KUKA KRL program: centerline_weld.src

&ACCESS RVO1
&REL 38
&COMMENT 03-10-R1 PNW1 NUT WELD
&PARAM TEMPLATE = C:\KRC\Roboter\Template\vorgabe
DEF CENTERLINE_WELD()
;********************************
; Gestamp Standards
; Line - BMW G65 (cell 03)
; Robot 03-10-R1 (BMW-03-10-R1-PNW1)
; Application - NUT WELD AT CENTERLINE PEDESTAL (ALL 3 NUTS)
;********************************
; PRODUCTION NUT WELD, CALLED BY style1app1opt1A..3B OUTSIDE DRY CYCLE WITH THE PART ALREADY
; AT THE WELD POSITION (NO ROBOT MOTION HERE): PEDESTAL START POSITION, UPPER PIN EXTEND,
; PART CLAMP CLOSE, GUN CLOSE, GUN STROKE CHECK (LPT), INTENSIFY, BOSCH WELD; THEN GUN
; OPEN, UPPER PIN RETRACT, PART CLAMP OPEN, LOWER PIN ADVANCE, QFP RETURN.
;WARNING: PEDESTAL ENTRY IS ONLY PARTLY CONFIRMED. THE CALLER CHECKS GUN OPEN (GUN_OPEN_CHECK) AND
;  MONITORS IT WITH INTERRUPTS 20-22; CLAMP OPEN AND QFP RETURNED ARE CHECKED BELOW ONLY AFTER THE
;  ROBOT IS ALREADY AT THE WELD POSITION (F01)
;NOTE: THE NUT IS NORMALLY PRELOADED BY PRELOAD() IN THE SUBMIT INTERPRETER (NUT_READY TRUE);
;  PRELOAD DRIVES THE SAME PEDESTAL VALVES, WITH NO OWNERSHIP BETWEEN THE TWO (F11)
;NOTE: DURING THIS WELD A FEED-ONLY PRELOAD STARTED BY WELD APPS 1-2 MAY BE FEEDING THE NEXT NUT
;  INTO THE SHUTTLE (NUTCYCLE_ACTIVE TRUE): THE FEED OUTPUT $OUT[476] IS LEFT TO IT (F52)
;NOTE: NO WATER FLOW CHECK BEFORE THE WELD (F09), NO FAULT CHECK AFTER THE WELD (F08),
;  NO TIMEOUT OR MESSAGE ON THE WAITS (F15), PIN POSITIONS NOT VERIFIED (F16)
;NOTE: NUT_READY IS NOT CLEARED WHEN THE NUT IS WELDED (F14)
;NOTE: NOTHING PUTS THE PEDESTAL IN A SAFE STATE IF THIS PROGRAM IS CANCELLED (F10)
;NOTE: USES $TIMER[14] (GUN-CLOSED TIMEOUT) AND $TIMER[15] (TIME IN THE WINDOW) (F26)
;NOTE: CL_CYCLE_TIME(2..13) RECORDS THE TIME OF EACH STEP ($TIMER[20], CL_CYCLE_TIME.dat) (F52)
;NOTE: LIMITS, PRESSURE WORDS AND WELD PROGRAM ARE CONSTANTS IN $config.dat (FOLD CENTERLINE CONTROL)
;********************************

;PEDESTAL REFERENCE VALUES - INFORMATION ONLY
;UPPER PIN POSITION CL_WeldPinPosition ($IN[591..606]) - NO PROGRAM READS IT (F16):
;UPPER PIN RETRACT =  27252      RANGE 26000 - 28000
;UPPER PIN EXTENDED = 6602       RANGE 6500- 7000
;UPPER PIN WELD POSITION = 11674 RANGE 10000 - 13500

;GUN STROKE CL_GunStrokePositionLPT ($IN[559..590], LPT):
;GUN RETRACT = 139815            RANGE 137000 - 142000  (CHECKED: GUN_OPEN_CHECK, nGunOpenMin..MAX)
;GUN EXTENDED = 61450            RANGE 60000 - 63000
;GUN WELD POSITION = 70915       RANGE 65000 - 76000    (CHECKED: CL_GUN_WELD_MIN..MAX = 69000..73000)

;ITV PRESSURE SET-POINT CL_GunPressureCmd ($OUT[506..521]):
;FORMULA CMD = (MPa / 0.9) * 4095
;CHECK: THIS TABLE IS NOT BYTE-SWAPPED. KRC_IO.xml SENDS THE WORD TO THE REGULATOR BYTE-SWAPPED,
;CHECK: AS ON R20 (THERE 0.30 MPa IS WRITTEN 21765). THIS PROGRAM WRITES CL_GUN_PRESS_BASE = 405 AND
;CHECK: CL_GUN_PRESS_WELD = 1820 (NOT SWAPPED) AND CL_GUN_PRESS_REST = 39425 AT THE END (SWAPPED
;CHECK: 0.09 MPa) - CONFIRM WHICH IS RIGHT ON THE ITV (F44)
;PRESSURE 455   0.10MPa    14.50 PSI
;PRESSURE 910   0.20MPa    29.01 PSI
;PRESSURE 1365  0.30MPa    43.51 PSI
;PRESSURE 1820  0.40MPa    58.02 PSI  (CL_GUN_PRESS_WELD)
;PRESSURE 2275  0.50MPa    72.52 PSI
;PRESSURE 2503  0.55MPa    79.77 PSI
;PRESSURE 2730  0.60MPa    87.02 PSI
;CL_GUN_PRESS_BASE = 405 = 0.089 MPa IF NOT SWAPPED

;CYCLE-TIME MARK - STEP 2 AT THE WELD POSITION (CL_CYCLE_TIME, F52)
CL_CYCLE_TIME(2)

;PEDESTAL START POSITION (NOT A FULL HOME: THE LOWER PIN IS ADVANCED)

;GUN OPEN - SIGNALS $OUT[472] dopw1_GunWork OFF, $OUT[471] dopw1_GunHome ON
dopw1_GunWork=FALSE
dopw1_GunHome=TRUE

;UPPER PIN RETRACT - SIGNALS $OUT[498] do498UpperPinExtend OFF, $OUT[499] do499UpperPinRetract ON
;CHECK: OLD COMMENT SAID UPPER PIN EXTEND; THE CODE RETRACTS THE UPPER PIN HERE (F27)
do498UpperPinExtend=FALSE
do499UpperPinRetract=TRUE

;PART CLAMP OPEN - SIGNALS $OUT[501] do501PartClampClose OFF, $OUT[502] do502PartClampOpen ON
do501PartClampClose=FALSE
do502PartClampOpen=TRUE
;WAIT PART CLAMP OPEN - SIGNAL $IN[466] di466PartClampOpen ON
WAIT FOR di466PartClampOpen

;LOWER PIN ADVANCE - SIGNALS $OUT[496] dopw1_ReturnPin OFF, $OUT[495] dopw1_AdvancePin ON
dopw1_ReturnPin=FALSE
dopw1_AdvancePin=TRUE

;QFP RETURN - SIGNALS $OUT[503] do503QFPAdvance OFF, $OUT[504] do504QFPReturn ON
do503QFPAdvance=FALSE
do504QFPReturn=TRUE
;WAIT QFP RETURNED - SIGNAL $IN[482] dipw1_SpearHome ON
WAIT FOR dipw1_SpearHome

;LOCAL NUT FEED - ONLY WHEN NO NUT WAS PRELOADED BY PRELOAD() (NUT_READY FALSE). NORMALLY
;  SKIPPED: PRELOAD SETS NUT_READY FOR EVERY NUT BEFORE THE CALLER MOVES IN
;NOTE: NOT WHILE A PRELOAD IS RUNNING (NUTCYCLE_ACTIVE): THE NEXT NUT MAY ALREADY BE IN THE SHUTTLE
;  (FEED-ONLY PRELOAD, F52). A RETRY AFTER THE GUN-CLOSED TIMEOUT THEN WELDS WITH WHAT IS ON THE
;  PIN; WITH NO NUT THE GUN-CLOSED CHECK STOPS AGAIN (F07)
IF NOT NUT_READY AND NOT NUTCYCLE_ACTIVE THEN
   ;LOWER PIN ADVANCE AND BLOW-OFF - SIGNALS $OUT[496] dopw1_ReturnPin OFF,
   ;  $OUT[495] dopw1_AdvancePin ON, $OUT[494] dopw1_BlowOff ON
   dopw1_ReturnPin=FALSE
   dopw1_AdvancePin=TRUE
   dopw1_BlowOff=TRUE

   ;QFP ADVANCE - SIGNALS $OUT[504] do504QFPReturn OFF, $OUT[503] do503QFPAdvance ON
   do504QFPReturn=FALSE
   do503QFPAdvance=TRUE
   ;WAIT QFP ADVANCED - SIGNAL $IN[470] di470QFPAdvanced ON
   WAIT FOR di470QFPAdvanced

   ;FEED NUT - SIGNAL $OUT[476] dopw1_StartFeed ON, THEN OFF, THEN WAIT 1.5 S
   ;NOTE: FEED COMPLETE CHECK $IN[481] dipw1_FeedComplt IS DISABLED (F25)
   ;CHECK: ON AND OFF BACK TO BACK IS A ZERO-LENGTH FEED PULSE; THE FEEDER MAY NEVER SEE IT (F25)
   dopw1_StartFeed=TRUE
   dopw1_StartFeed=FALSE
   WAIT SEC 1.5
   ;BLOW-OFF OFF - SIGNAL $OUT[494] dopw1_BlowOff OFF
   dopw1_BlowOff=FALSE

   ;QFP RETURN - SIGNALS $OUT[503] do503QFPAdvance OFF, $OUT[504] do504QFPReturn ON
   do503QFPAdvance=FALSE
   do504QFPReturn=TRUE
   ;WAIT QFP RETURNED - SIGNAL $IN[482] dipw1_SpearHome ON
   WAIT FOR dipw1_SpearHome
ENDIF
;CYCLE-TIME MARK - STEP 3 PEDESTAL READY (CL_CYCLE_TIME, F52)
CL_CYCLE_TIME(3)

;UPPER PIN EXTEND - SIGNALS $OUT[499] do499UpperPinRetract OFF, $OUT[498] do498UpperPinExtend ON
do499UpperPinRetract=FALSE
do498UpperPinExtend=TRUE

;GUN GENERAL PRESSURE - SIGNALS $OUT[506..521] CL_GunPressureCmd = CL_GUN_PRESS_BASE (F44)
CL_GunPressureCmd=CL_GUN_PRESS_BASE

;RESET BOSCH HANDSHAKE - SIGNALS $OUT[483] dopw1_WeldInit OFF, $OUT[481] dopw1_WeldContactEnable OFF,
;  $OUT[482] dopw1_WeldOnExternal OFF, $OUT[486..493] gdopw1_SpotNumber = 0
dopw1_WeldInit=FALSE
dopw1_WeldContactEnable=FALSE
dopw1_WeldOnExternal=FALSE
gdopw1_SpotNumber=0
;RESET PEDESTAL OUTPUTS - SIGNALS $OUT[494] dopw1_BlowOff OFF,
;  $OUT[474] dopw1_Nut1Intensify OFF (NOT ON THE BUS), $OUT[473] dopw1_Nut1Intensify_Home ON
dopw1_Nut1Intensify=FALSE
dopw1_Nut1Intensify_Home=TRUE
dopw1_BlowOff=FALSE
;FEED OFF - SIGNAL $OUT[476] dopw1_StartFeed OFF, ONLY WHEN NO PRELOAD IS RUNNING: A PRELOAD STARTED
;  BY THE WELD APP (NUT_FEED_START) FEEDS THE NEXT NUT INTO THE SHUTTLE DURING THIS WELD (F52)
IF NOT NUTCYCLE_ACTIVE THEN
   dopw1_StartFeed=FALSE
ENDIF
;GUN GENERAL PRESSURE AGAIN - SIGNALS $OUT[506..521] CL_GunPressureCmd = CL_GUN_PRESS_BASE
CL_GunPressureCmd=CL_GUN_PRESS_BASE
;ENABLE BOSCH WELD TIMER - SIGNALS $OUT[481] dopw1_WeldContactEnable ON,
;  $OUT[482] dopw1_WeldOnExternal ON
dopw1_WeldContactEnable=TRUE
dopw1_WeldOnExternal=TRUE

;WAIT BOSCH READY - SIGNAL $IN[484] dipw1_Ready ON
WAIT FOR dipw1_Ready
;CYCLE-TIME MARK - STEP 4 BOSCH READY (CL_CYCLE_TIME, F52)
CL_CYCLE_TIME(4)

;PART CLAMP CLOSE - SIGNALS $OUT[502] do502PartClampOpen OFF, $OUT[501] do501PartClampClose ON
do502PartClampOpen=FALSE
do501PartClampClose=TRUE
;WAIT PART CLAMP CLOSED - SIGNAL $IN[467] di467PartClampClosed ON
WAIT FOR di467PartClampClosed
;CYCLE-TIME MARK - STEP 5 PART CLAMP CLOSED (CL_CYCLE_TIME, F52)
CL_CYCLE_TIME(5)

;GUN CLOSE - SIGNALS $OUT[471] dopw1_GunHome OFF, WAIT 0.2 S, $OUT[472] dopw1_GunWork ON
dopw1_GunHome=FALSE
WAIT SEC 0.2
dopw1_GunWork=TRUE

;LOWER PIN BOTH VALVES OFF (OLD COMMENT: REMOVE AIR FROM THE LOWER PIN) -
;  SIGNALS $OUT[495] dopw1_AdvancePin OFF, $OUT[496] dopw1_ReturnPin OFF
dopw1_AdvancePin=FALSE
dopw1_ReturnPin=FALSE

;CONFIRM GUN CLOSED: CL_GunStrokePositionLPT IN CL_GUN_WELD_MIN..CL_GUN_WELD_MAX WITHOUT A BREAK
;  FOR CL_GUN_IN_WINDOW_TIME MS ($TIMER[15]), WITHIN CL_GUN_CLOSE_TIMEOUT MS ($TIMER[14])
;START BOTH TIMERS
$TIMER_STOP[14]=TRUE
$TIMER[14]=0
$TIMER_STOP[14]=FALSE
$TIMER_STOP[15]=TRUE
$TIMER[15]=0
$TIMER_STOP[15]=FALSE

LOOP
   IF (CL_GunStrokePositionLPT>=CL_GUN_WELD_MIN) AND (CL_GunStrokePositionLPT<=CL_GUN_WELD_MAX) THEN
      ;IN THE WINDOW LONG ENOUGH: GUN CLOSED ON THE NUT
      IF $TIMER[15]>=CL_GUN_IN_WINDOW_TIME THEN
         EXIT
      ENDIF
   ELSE
      ;OUT OF THE WINDOW: RESTART THE TIME IN THE WINDOW
      $TIMER_STOP[15]=TRUE
      $TIMER[15]=0
      $TIMER_STOP[15]=FALSE

      ;TIMEOUT: NUT_READY=FALSE AND HALT
      IF $TIMER[14]>=CL_GUN_CLOSE_TIMEOUT THEN
         $TIMER_STOP[14]=TRUE
         $TIMER[14]=0
         $TIMER_STOP[15]=TRUE
         $TIMER[15]=0
         NUT_READY=FALSE
         ;WARNING: HALT WITH NO MESSAGE IS STILL THE ONLY FAULT HANDLING - A DIALOG THAT NAMES THE
         ;  FAULT (NO NUT / DOUBLE NUT / GUN NOT CLOSED) WITH RETRY AND ABORT IS STILL TO DO (F07)
         HALT
         ;AFTER THE RESUME: RESTART BOTH TIMERS, SO THE CHECK TIMES OUT AGAIN IF THE GUN IS STILL
         ;  NOT CLOSED (F07)
         $TIMER_STOP[14]=FALSE
         $TIMER_STOP[15]=FALSE
      ENDIF
   ENDIF
ENDLOOP

;GUN CLOSED: STOP AND CLEAR BOTH TIMERS
$TIMER_STOP[14]=TRUE
$TIMER[14]=0
$TIMER_STOP[15]=TRUE
$TIMER[15]=0
;CYCLE-TIME MARK - STEP 6 GUN CLOSED ON THE NUT (CL_CYCLE_TIME, F52)
CL_CYCLE_TIME(6)

;WELD ON EXTERNAL - SIGNAL $OUT[482] dopw1_WeldOnExternal ON (ALREADY ON SINCE THE BOSCH ENABLE)
dopw1_WeldOnExternal=TRUE

;SELECT THE WELD PROGRAM - SIGNALS $OUT[486..493] gdopw1_SpotNumber = CL_WELD_PROGRAM (2)
;CHECK: OLD COMMENT SAID SCHEDULE 7; THE CODE SELECTS PROGRAM 2 - CONFIRM ON THE BOSCH TIMER (F27)
gdopw1_SpotNumber=CL_WELD_PROGRAM

;WAIT BOSCH READY - SIGNAL $IN[484] dipw1_Ready ON
WAIT FOR dipw1_Ready
;CYCLE-TIME MARK - STEP 7 BOSCH READY AGAIN (CL_CYCLE_TIME, F52)
CL_CYCLE_TIME(7)

;INTENSIFY - GUN PRESSURE - SIGNALS $OUT[506..521] CL_GunPressureCmd = CL_GUN_PRESS_WELD (F44)
CL_GunPressureCmd=CL_GUN_PRESS_WELD

;INTENSIFY - SIGNALS $OUT[494] dopw1_BlowOff ON, $OUT[473] dopw1_Nut1Intensify_Home OFF,
;  $OUT[474] dopw1_Nut1Intensify ON (NOT MAPPED TO THE BUS, NO EFFECT)
dopw1_BlowOff=TRUE
dopw1_Nut1Intensify_Home=FALSE
dopw1_Nut1Intensify=TRUE

;WAIT INTENSIFY PRESSURE OK - SIGNAL $IN[479] dipw1_IntensfPresOk ON (NO TIMEOUT, F15)
WAIT FOR dipw1_IntensfPresOk
;CYCLE-TIME MARK - STEP 8 INTENSIFY PRESSURE OK (CL_CYCLE_TIME, F52)
CL_CYCLE_TIME(8)

;CONFIRM GUN POSITION BEFORE WELDING - WAIT CL_GunStrokePositionLPT IN CL_GUN_WELD_MIN..MAX
WAIT FOR (CL_GunStrokePositionLPT>=CL_GUN_WELD_MIN) AND (CL_GunStrokePositionLPT<=CL_GUN_WELD_MAX)

;WELD - SIGNAL $OUT[483] dopw1_WeldInit ON, WAIT $IN[483] dipw1_WeldComplete ON
dopw1_WeldInit=TRUE

WAIT FOR dipw1_WeldComplete
;CYCLE-TIME MARK - STEP 9 WELD COMPLETE ON (CL_CYCLE_TIME, F52)
CL_CYCLE_TIME(9)

;WELD START OFF - SIGNAL $OUT[483] dopw1_WeldInit OFF, WAIT $IN[483] dipw1_WeldComplete OFF
dopw1_WeldInit=FALSE
WAIT FOR NOT dipw1_WeldComplete
;CYCLE-TIME MARK - STEP 10 WELD COMPLETE OFF (CL_CYCLE_TIME, F52)
CL_CYCLE_TIME(10)
;NOTE: NO FAULT CHECK AFTER THE WELD - $IN[485] dipw1_Fault IS NOT READ BY ANY ACTIVE CODE
;  (ONLY BY THE UNUSED NUTWELD AND DISABLED AUTOMATIONCORE ROUTINES); WELD COMPLETE
;  IS TAKEN AS A GOOD WELD (F08)

;RELEASE INTENSIFY - SIGNALS $OUT[474] dopw1_Nut1Intensify OFF,
;  $OUT[473] dopw1_Nut1Intensify_Home ON, $OUT[494] dopw1_BlowOff OFF
dopw1_Nut1Intensify=FALSE
dopw1_Nut1Intensify_Home=TRUE
dopw1_BlowOff=FALSE

;GUN GENERAL PRESSURE - SIGNALS $OUT[506..521] CL_GunPressureCmd = CL_GUN_PRESS_BASE (F44)
CL_GunPressureCmd=CL_GUN_PRESS_BASE

;CLEAR WELD PROGRAM NUMBER - SIGNALS $OUT[486..493] gdopw1_SpotNumber = 0
gdopw1_SpotNumber=0

;STOP THE GUN-CLOSED TIMER $TIMER[14]
$TIMER_STOP[14]=TRUE
$TIMER[14]=0

;GUN OPEN - SIGNALS $OUT[472] dopw1_GunWork OFF, WAIT 0.2 S, $OUT[471] dopw1_GunHome ON
dopw1_GunWork=FALSE
WAIT SEC 0.2
dopw1_GunHome=TRUE

;GUN OPEN INTERLOCK BEFORE THE PART IS RELEASED AND THE ROBOT LEAVES - GUN_OPEN_CHECK: SUBMIT RUNNING,
;WATER OK, CL_GunStrokePositionLPT IN 137000..142000 (MESSAGE AFTER 2 S, WAITS), THEN 0.2 S (F01)
GUN_OPEN_CHECK()
;CYCLE-TIME MARK - STEP 11 GUN OPEN CONFIRMED (CL_CYCLE_TIME, F52)
CL_CYCLE_TIME(11)
WAIT SEC 0.2

;UPPER PIN RETRACT - SIGNALS $OUT[498] do498UpperPinExtend OFF, $OUT[499] do499UpperPinRetract ON
do498UpperPinExtend=FALSE
do499UpperPinRetract=TRUE

;PART CLAMP OPEN - SIGNALS $OUT[501] do501PartClampClose OFF, $OUT[502] do502PartClampOpen ON
do501PartClampClose=FALSE
do502PartClampOpen=TRUE
;WAIT PART CLAMP OPEN - SIGNAL $IN[466] di466PartClampOpen ON
WAIT FOR di466PartClampOpen
;CYCLE-TIME MARK - STEP 12 PART CLAMP OPEN (CL_CYCLE_TIME, F52)
CL_CYCLE_TIME(12)

;LOWER PIN ADVANCE - SIGNALS $OUT[496] dopw1_ReturnPin OFF, $OUT[495] dopw1_AdvancePin ON
;CHECK: OLD COMMENT SAID LOWER PIN RETURN; THE CODE ADVANCES THE PIN HERE (F27)
dopw1_ReturnPin=FALSE
dopw1_AdvancePin=TRUE

;QFP RETURN - SIGNALS $OUT[503] do503QFPAdvance OFF, $OUT[504] do504QFPReturn ON
do503QFPAdvance=FALSE
do504QFPReturn=TRUE
;WAIT QFP RETURNED - SIGNAL $IN[482] dipw1_SpearHome ON
WAIT FOR dipw1_SpearHome

;FINAL RESET - SIGNALS $OUT[483] dopw1_WeldInit OFF, $OUT[486..493] gdopw1_SpotNumber = 0
dopw1_WeldInit=FALSE
gdopw1_SpotNumber=0
;FEED OFF - SIGNAL $OUT[476] dopw1_StartFeed OFF, ONLY WHEN NO PRELOAD IS RUNNING (AS ABOVE, F52)
IF NOT NUTCYCLE_ACTIVE THEN
   dopw1_StartFeed=FALSE
ENDIF

;CHECK: CL_GUN_PRESS_REST (39425) BELOW IS THE R20 BYTE-SWAPPED 0.09 MPa, NOT THE CL_GUN_PRESS_BASE
;CHECK: USED ABOVE; NOT SWAPPED IT IS OUT OF THE ITV RANGE (0..4095). THE GUN RESTS AT THIS VALUE
;CHECK: UNTIL THE NEXT WELD (F44)
;INTENSIFY OFF - SIGNALS $OUT[474] dopw1_Nut1Intensify OFF,
;  $OUT[473] dopw1_Nut1Intensify_Home ON, $OUT[494] dopw1_BlowOff OFF
dopw1_Nut1Intensify=FALSE
dopw1_Nut1Intensify_Home=TRUE
dopw1_BlowOff=FALSE
;REST PRESSURE - SIGNALS $OUT[506..521] CL_GunPressureCmd = CL_GUN_PRESS_REST (39425)
CL_GunPressureCmd=CL_GUN_PRESS_REST

;BOSCH DISABLE - SIGNALS $OUT[481] dopw1_WeldContactEnable OFF, $OUT[482] dopw1_WeldOnExternal OFF
dopw1_WeldContactEnable=FALSE
dopw1_WeldOnExternal=FALSE

;CYCLE-TIME MARK - STEP 13 CENTERLINE_WELD ENDS (CL_CYCLE_TIME, F52)
CL_CYCLE_TIME(13)
END
